(* Logix 5000 project; controller Final vendor 1 type 14 code 242 rev 32.11; software revision 32.00 *)

TASK MainTask (continuous, watchdog 500 ms) : MainProgram
TASK SafetyTask (periodic, rate 20 ms, priority 10, watchdog 20 ms, safety) : SafetyProgram

MODULES
   Local : vendor 1 type 14 code 242 (5069 0, rev 32.11)
      IO_002 : 5069-IF8 (5069 2, rev 2.1, StandardDataDriven RPI 100 ms)
      IO_001 : 5069-IF8 (5069 1, rev 2.1, StandardDataDriven RPI 100 ms)
      IO_003 : 5069-IF8 (5069 3, rev 2.1, StandardDataDriven RPI 100 ms)
      IO_006 : vendor 1 type 7 code 394 (5069 6, rev 2.1, StandardDataDriven RPI 5 ms)
      IO_004 : vendor 1 type 7 code 395 (5069 4, rev 2.1, StandardDataDriven RPI 5 ms)
      IO_005 : vendor 1 type 7 code 395 (5069 5, rev 2.1, StandardDataDriven RPI 5 ms)
      IO_007 : vendor 1 type 109 code 90 (5069 7, rev 3.1, StandardDataDriven RPI 80 ms)
      EN_001 : 1734-AENTR (Ethernet 192.168.1.60, rev 5.1, Output RPI 20 ms)
         EN_004 : 1734-485ASC (PointIO 3, rev 4.1, Output RPI 80 ms)
         EN_003 : vendor 1 type 35 code 16 (PointIO 2, rev 2.1, Input RPI 10 ms, Output RPI 20 ms)
         EN_002 : vendor 1 type 35 code 15 (PointIO 1, rev 2.1, Input RPI 10 ms)
END_MODULES

TYPE ASC_module_string :
STRUCT
   LEN : DINT;
   DATA : SINT[100];
END_STRUCT
END_TYPE

TYPE SensorType :   // To monitor the sensor readings, we use this data type
STRUCT
   CurrentValue : DINT;
   PreviousValue0 : DINT;
   PreviousValue1 : DINT;
   PreviousValue2 : DINT;
   PreviousValue3 : DINT;
   PreviousValue4 : DINT;
   PreviousValue5 : DINT;
   PreviousValue6 : DINT;
   PreviousValue7 : DINT;
   PreviousValue8 : DINT;
   PreviousValue9 : DINT;
   Mean10 : DINT;
   StanDev : DINT;
   State : DINT;
   Count : DINT;
   MeanStart : BOOL;
END_STRUCT
END_TYPE

TYPE String122 :
STRUCT
   LEN : DINT;
   DATA : SINT[122];
END_STRUCT
END_TYPE

VAR_GLOBAL   (* controller tags *)
   ACC_TIMER : DINT;
   ASC_module_Data : ASC_module_string;
   AT : BOOL;
   B0_Max : DINT;
   B0_Min : DINT;
   B1_Max : DINT;
   B1_Min : DINT;
   B3_Max : DINT;
   B3_Min : DINT;
   B_Check : BOOL;
   B_Checked : BOOL;
   B_NomCount : DINT := 24;
   B_Pres0 : SensorType := (CurrentValue := 15, PreviousValue0 := 15, PreviousValue1 := 15, PreviousValue2 := 15, PreviousValue3 := 15, PreviousValue4 := 15, PreviousValue5 := 15, PreviousValue6 := 15, PreviousValue7 := 15, PreviousValue8 := 15, PreviousValue9 := 15, Mean10 := 15, Count := 7, MeanStart := 1);   // Holds all values related to Brakes Pressure Sensor #0
   B_Pres1 : SensorType := (CurrentValue := 15, PreviousValue0 := 15, PreviousValue1 := 15, PreviousValue2 := 15, PreviousValue3 := 15, PreviousValue4 := 15, PreviousValue5 := 15, PreviousValue6 := 15, PreviousValue7 := 15, PreviousValue8 := 15, PreviousValue9 := 15, Mean10 := 15, Count := 7, MeanStart := 1);   // Holds all values related to Brakes Pressure Sensor #1
   B_Pres2 : SensorType := (CurrentValue := 15, PreviousValue0 := 15, PreviousValue1 := 15, PreviousValue2 := 15, PreviousValue3 := 15, PreviousValue4 := 15, PreviousValue5 := 15, PreviousValue6 := 15, PreviousValue7 := 15, PreviousValue8 := 15, PreviousValue9 := 15, Mean10 := 15, Count := 7, MeanStart := 1);   // Holds all values related to Brakes Pressure Sensor #2
   B_Pres3 : SensorType := (CurrentValue := 15, PreviousValue0 := 15, PreviousValue1 := 15, PreviousValue2 := 15, PreviousValue3 := 15, PreviousValue4 := 15, PreviousValue5 := 15, PreviousValue6 := 15, PreviousValue7 := 15, PreviousValue8 := 15, PreviousValue9 := 15, Mean10 := 15, Count := 7, MeanStart := 1);   // Holds all values related to Brakes Pressure Sensor #3
   B_Pres4 : SensorType := (CurrentValue := 15, PreviousValue0 := 15, PreviousValue1 := 15, PreviousValue2 := 15, PreviousValue3 := 15, PreviousValue4 := 15, PreviousValue5 := 15, PreviousValue6 := 15, PreviousValue7 := 15, PreviousValue8 := 15, PreviousValue9 := 15, Mean10 := 15, Count := 7, MeanStart := 1);   // Holds all values related to Brakes Pressure Sensor #4
   B_Pres5 : SensorType := (CurrentValue := 15, PreviousValue0 := 15, PreviousValue1 := 15, PreviousValue2 := 15, PreviousValue3 := 15, PreviousValue4 := 15, PreviousValue5 := 15, PreviousValue6 := 15, PreviousValue7 := 15, PreviousValue8 := 15, PreviousValue9 := 15, Mean10 := 15, Count := 7, MeanStart := 1);   // Holds all values related to Brakes Pressure Sensor #5
   B_Pres6 : SensorType := (CurrentValue := 15, PreviousValue0 := 15, PreviousValue1 := 15, PreviousValue2 := 15, PreviousValue3 := 15, PreviousValue4 := 15, PreviousValue5 := 15, PreviousValue6 := 15, PreviousValue7 := 15, PreviousValue8 := 15, PreviousValue9 := 15, Mean10 := 15, Count := 7, MeanStart := 1);   // Holds all values related to Brakes Pressure Sensor #6
   B_Pres7 : SensorType := (CurrentValue := 15, PreviousValue0 := 15, PreviousValue1 := 15, PreviousValue2 := 15, PreviousValue3 := 15, PreviousValue4 := 15, PreviousValue5 := 15, PreviousValue6 := 15, PreviousValue7 := 15, PreviousValue8 := 15, PreviousValue9 := 15, Mean10 := 15, Count := 7, MeanStart := 1);   // Holds all values related to Brakes Pressure Sensor #7
   B_Pres8 : SensorType := (CurrentValue := 15, PreviousValue0 := 15, PreviousValue1 := 15, PreviousValue2 := 15, PreviousValue3 := 15, PreviousValue4 := 15, PreviousValue5 := 15, PreviousValue6 := 15, PreviousValue7 := 15, PreviousValue8 := 15, PreviousValue9 := 15, Mean10 := 15, Count := 7, MeanStart := 1);   // Holds all values related to Brakes Pressure Sensor #8
   B_Pres9 : SensorType := (CurrentValue := 15, PreviousValue0 := 15, PreviousValue1 := 15, PreviousValue2 := 15, PreviousValue3 := 15, PreviousValue4 := 15, PreviousValue5 := 15, PreviousValue6 := 15, PreviousValue7 := 15, PreviousValue8 := 15, PreviousValue9 := 15, Mean10 := 15, Count := 7, MeanStart := 1);   // Holds all values related to Brakes Pressure Sensor #9
   B_Tem0 : SensorType := (CurrentValue := 92, PreviousValue0 := 92, PreviousValue1 := 92, PreviousValue2 := 92, PreviousValue3 := 92, PreviousValue4 := 92, PreviousValue5 := 92, PreviousValue6 := 92, PreviousValue7 := 92, PreviousValue8 := 92, PreviousValue9 := 92, Mean10 := 92, Count := 7, MeanStart := 1);   // Holds all values related to Brakes Temperature Sensor #0
   B_Tem1 : SensorType := (CurrentValue := 92, PreviousValue0 := 92, PreviousValue1 := 92, PreviousValue2 := 92, PreviousValue3 := 92, PreviousValue4 := 92, PreviousValue5 := 92, PreviousValue6 := 92, PreviousValue7 := 92, PreviousValue8 := 92, PreviousValue9 := 92, Mean10 := 92, Count := 7, MeanStart := 1);   // Holds all values related to Brakes Temperature Sensor #1
   Bat_Amp_State : DINT;
   BAT_FLAG : BOOL;
   Bat_Temp_State : DINT;
   Bat_Volt_State : DINT;
   BatCurrent_Pre : STRING;
   BatTemp_Pre : STRING;
   BATTERY_CHARGE : REAL := 104.21566;
   BATTERY_CURRENT : DINT;
   BATTERY_TEMP : REAL := 304.73172;
   BATTERY_VOLTAGE : REAL := 29.25294;
   BatteryA : REAL := 0.00112924;
   BatteryB : REAL := 0.000234108;
   BatteryC : REAL := 8.7755e-08;
   BatteryCommand : STRING := ':0102A0000EF6~';
   BatVoltage_Pre : STRING;
   BCount : DINT;
   bfr_SysSec : DINT := 58;
   BPCount : DINT;
   BRAKE_FLAG : BOOL;
   BRAKE_SUBSTATE1 : DINT;
   BRAKE_SUBSTATE2 : DINT;
   BRAKE_TIMER : FBD_TIMER;
   BRPM : DINT;
   BT : BOOL;
   C_Las0 : SensorType := (CurrentValue := 213, PreviousValue0 := 213, PreviousValue1 := 213, PreviousValue2 := 213, PreviousValue3 := 213, PreviousValue4 := 213, PreviousValue5 := 213, PreviousValue6 := 213, PreviousValue7 := 213, PreviousValue8 := 213, PreviousValue9 := 213, Mean10 := 213, Count := 7, MeanStart := 1);   // Holds all values related to Controls Laser Sensor #0
   C_Las1 : SensorType := (CurrentValue := 177, PreviousValue0 := 177, PreviousValue1 := 177, PreviousValue2 := 177, PreviousValue3 := 177, PreviousValue4 := 177, PreviousValue5 := 177, PreviousValue6 := 177, PreviousValue7 := 177, PreviousValue8 := 177, PreviousValue9 := 177, Mean10 := 177, Count := 7, MeanStart := 1);   // Holds all values related to Controls Laser Sensor #1
   CA : BOOL := 1;
   CB : BOOL;
   CC : BOOL;
   CD1 : BOOL := 1;
   CD2 : BOOL := 1;
   CD3 : BOOL := 1;
   COAST_TIMER : DINT;
   COAST_TONR : DINT;
   COMMAND : DINT := 1;
   COMN_FLAG : BOOL;
   ConversionResistance : REAL := 7533.3335;
   ConversionVoltage : REAL := 3.0;
   count : DINT;
   COUNT_LAS0 : DINT := 213;
   COUNT_LAS1 : DINT := 177;
   CP1 : BOOL := 1;
   CP2 : BOOL;
   CPX : BOOL;
   CT : BOOL;
   Current_OoR : BOOL := 1;
   CurrentState : DINT;
   CV : BOOL;
   DualStop : BOOL;
   EStop : BOOL;
   Initialized : DINT := 5380;
   InverseTemp : REAL := 0.003281575;
   LastValue : DINT;
   LastValue0 : DINT;
   LastValue1 : DINT;
   LenOut : SINT := 14;
   Limit1 : BOOL;
   Limit2 : BOOL;
   Local_TONR : FBD_TIMER;
   LogR : REAL := 8.927093;
   LSD_AA : BOOL;
   LSD_DR : BOOL;
   LSD_FR : BOOL;
   LSD_LC : DINT;
   LSD_PWR : BOOL;
   Mask : DINT := 16#0000_000f;
   my_TONR : FBD_TIMER;
   P_Check : DINT;
   P_Max : DINT;
   P_Mean : DINT;
   P_Min : DINT;
   P_NomCount : DINT := 20;
   P_Pres0 : SensorType := (CurrentValue := -16, PreviousValue0 := -16, PreviousValue1 := -16, PreviousValue2 := -16, PreviousValue3 := -16, PreviousValue4 := -16, PreviousValue5 := -16, PreviousValue6 := -16, PreviousValue7 := -16, PreviousValue8 := -16, PreviousValue9 := -16, Mean10 := -16, Count := 7, MeanStart := 1);   // Holds all values related to Pressure Pressure Sensor #0
   P_Pres0_FAILURE : BOOL;
   P_Pres1 : SensorType := (CurrentValue := -312, PreviousValue0 := -312, PreviousValue1 := -312, PreviousValue2 := -312, PreviousValue3 := -312, PreviousValue4 := -312, PreviousValue5 := -312, PreviousValue6 := -312, PreviousValue7 := -312, PreviousValue8 := -312, PreviousValue9 := -312, Count := 7);   // Holds all values related to Pressure Pressure Sensor #1
   P_Pres1_FAILURE : BOOL;
   P_Pres2 : SensorType := (CurrentValue := -312, PreviousValue0 := -312, PreviousValue1 := -312, PreviousValue2 := -312, PreviousValue3 := -312, PreviousValue4 := -312, PreviousValue5 := -312, PreviousValue6 := -312, PreviousValue7 := -312, PreviousValue8 := -312, PreviousValue9 := -312, Mean10 := -312, Count := 7, MeanStart := 1);   // Holds all values related to Pressure Pressure Sensor #2
   P_Pres2_FAILURE : BOOL;
   P_Pres3 : SensorType := (CurrentValue := -312, PreviousValue0 := -312, PreviousValue1 := -312, PreviousValue2 := -312, PreviousValue3 := -312, PreviousValue4 := -312, PreviousValue5 := -312, PreviousValue6 := -312, PreviousValue7 := -312, PreviousValue8 := -312, PreviousValue9 := -312, Mean10 := -312, Count := 7, MeanStart := 1);
   P_Pres3_FAILURE : BOOL;
   P_Pres4 : SensorType := (CurrentValue := -312, PreviousValue0 := -312, PreviousValue1 := -312, PreviousValue2 := -312, PreviousValue3 := -312, PreviousValue4 := -312, PreviousValue5 := -312, PreviousValue6 := -312, PreviousValue7 := -312, PreviousValue8 := -312, PreviousValue9 := -312, Mean10 := -312, Count := 7, MeanStart := 1);
   P_Pres4_FAILURE : BOOL;
   P_Tem0 : SensorType;   // Holds all values related to Pressure Temperature Sensor #0
   P_Tem0_FAILURE : BOOL;
   P_Tem1 : SensorType := (CurrentValue := 93, PreviousValue0 := 93, PreviousValue1 := 93, PreviousValue2 := 93, PreviousValue3 := 93, PreviousValue4 := 93, PreviousValue5 := 93, PreviousValue6 := 93, PreviousValue7 := 93, PreviousValue8 := 93, PreviousValue9 := 93, Mean10 := 93, Count := 7, MeanStart := 1);   // Holds all values related to Pressure Temperature Sensor #1
   P_Tem1_FAILURE : BOOL;
   P_Tem2 : SensorType := (CurrentValue := 93, PreviousValue0 := 93, PreviousValue1 := 93, PreviousValue2 := 93, PreviousValue3 := 93, PreviousValue4 := 93, PreviousValue5 := 93, PreviousValue6 := 93, PreviousValue7 := 93, PreviousValue8 := 93, PreviousValue9 := 93, Mean10 := 93, Count := 7, MeanStart := 1);
   P_Tem2_FAILURE : BOOL;
   P_Tem3 : SensorType := (CurrentValue := 93, PreviousValue0 := 93, PreviousValue1 := 93, PreviousValue2 := 93, PreviousValue3 := 93, PreviousValue4 := 93, PreviousValue5 := 93, PreviousValue6 := 93, PreviousValue7 := 93, PreviousValue8 := 93, PreviousValue9 := 93, Mean10 := 93, Count := 7, MeanStart := 1);
   P_Tem3_FAILURE : BOOL;
   P_Tem4 : SensorType := (CurrentValue := 93, PreviousValue0 := 93, PreviousValue1 := 93, PreviousValue2 := 93, PreviousValue3 := 93, PreviousValue4 := 93, PreviousValue5 := 93, PreviousValue6 := 93, PreviousValue7 := 93, PreviousValue8 := 93, PreviousValue9 := 93, Mean10 := 93, Count := 7, MeanStart := 1);
   P_Tem4_FAILURE : BOOL;
   POD_ACCELERATION : DINT;
   POD_DISTANCE : DINT := 1185672;
   POD_TIME : DINT[2] := ([0] := -1035744607, [1] := 205981);
   POD_VELOCITY : DINT;
   PREV_ACCELERATION : DINT;
   PREV_DISTANCE : DINT := 1185672;
   PREV_TIME : DINT[2] := ([0] := -1035744799);
   PREV_VELOCITY : DINT;
   PROP_FLAG : BOOL;
   PROP_STATE : BOOL;
   PROP_TNK_PRES : DINT;
   RcvRecord : SINT := 1;
   READY : BOOL;
   RxData : String122;
   RxID : SINT := 1;
   S_B_Pres0 : SensorType := (CurrentValue := 15, PreviousValue0 := 15, PreviousValue1 := 15, PreviousValue2 := 15, PreviousValue3 := 15, PreviousValue4 := 15, PreviousValue5 := 15, PreviousValue6 := 15, PreviousValue7 := 15, PreviousValue8 := 15, PreviousValue9 := 15, Mean10 := 15, Count := 7, MeanStart := 1);
   S_B_Pres1 : SensorType := (CurrentValue := 15, PreviousValue0 := 15, PreviousValue1 := 15, PreviousValue2 := 15, PreviousValue3 := 15, PreviousValue4 := 15, PreviousValue5 := 15, PreviousValue6 := 15, PreviousValue7 := 15, PreviousValue8 := 15, PreviousValue9 := 15, Mean10 := 15, Count := 7, MeanStart := 1);
   S_B_Pres2 : SensorType := (CurrentValue := 15, PreviousValue0 := 15, PreviousValue1 := 15, PreviousValue2 := 15, PreviousValue3 := 15, PreviousValue4 := 15, PreviousValue5 := 15, PreviousValue6 := 15, PreviousValue7 := 15, PreviousValue8 := 15, PreviousValue9 := 15, Mean10 := 15, Count := 7, MeanStart := 1);
   S_B_Pres3 : SensorType := (CurrentValue := 15, PreviousValue0 := 15, PreviousValue1 := 15, PreviousValue2 := 15, PreviousValue3 := 15, PreviousValue4 := 15, PreviousValue5 := 15, PreviousValue6 := 15, PreviousValue7 := 15, PreviousValue8 := 15, PreviousValue9 := 15, Mean10 := 15, Count := 7, MeanStart := 1);
   S_B_Pres4 : SensorType := (CurrentValue := 15, PreviousValue0 := 15, PreviousValue1 := 15, PreviousValue2 := 15, PreviousValue3 := 15, PreviousValue4 := 15, PreviousValue5 := 15, PreviousValue6 := 15, PreviousValue7 := 15, PreviousValue8 := 15, PreviousValue9 := 15, Mean10 := 15, Count := 7, MeanStart := 1);
   S_B_Pres5 : SensorType := (CurrentValue := 15, PreviousValue0 := 15, PreviousValue1 := 15, PreviousValue2 := 15, PreviousValue3 := 15, PreviousValue4 := 15, PreviousValue5 := 15, PreviousValue6 := 15, PreviousValue7 := 15, PreviousValue8 := 15, PreviousValue9 := 15, Mean10 := 15, Count := 7, MeanStart := 1);
   S_B_Pres6 : SensorType := (CurrentValue := 15, PreviousValue0 := 15, PreviousValue1 := 15, PreviousValue2 := 15, PreviousValue3 := 15, PreviousValue4 := 15, PreviousValue5 := 15, PreviousValue6 := 15, PreviousValue7 := 15, PreviousValue8 := 15, PreviousValue9 := 15, Mean10 := 15, Count := 7, MeanStart := 1);
   S_B_Pres7 : SensorType := (CurrentValue := 15, PreviousValue0 := 15, PreviousValue1 := 15, PreviousValue2 := 15, PreviousValue3 := 15, PreviousValue4 := 15, PreviousValue5 := 15, PreviousValue6 := 15, PreviousValue7 := 15, PreviousValue8 := 15, PreviousValue9 := 15, Mean10 := 15, Count := 7, MeanStart := 1);
   S_B_Pres8 : SensorType := (CurrentValue := 15, PreviousValue0 := 15, PreviousValue1 := 15, PreviousValue2 := 15, PreviousValue3 := 15, PreviousValue4 := 15, PreviousValue5 := 15, PreviousValue6 := 15, PreviousValue7 := 15, PreviousValue8 := 15, PreviousValue9 := 15, Mean10 := 15, Count := 7, MeanStart := 1);
   S_B_Pres9 : SensorType := (CurrentValue := 15, PreviousValue0 := 15, PreviousValue1 := 15, PreviousValue2 := 15, PreviousValue3 := 15, PreviousValue4 := 15, PreviousValue5 := 15, PreviousValue6 := 15, PreviousValue7 := 15, PreviousValue8 := 15, PreviousValue9 := 15, Mean10 := 15, Count := 7, MeanStart := 1);
   S_B_Tem0 : SensorType := (CurrentValue := 92, PreviousValue0 := 92, PreviousValue1 := 92, PreviousValue2 := 92, PreviousValue3 := 92, PreviousValue4 := 92, PreviousValue5 := 92, PreviousValue6 := 92, PreviousValue7 := 92, PreviousValue8 := 92, PreviousValue9 := 92, Mean10 := 92, Count := 7, MeanStart := 1);
   S_B_Tem1 : SensorType := (CurrentValue := 92, PreviousValue0 := 92, PreviousValue1 := 92, PreviousValue2 := 92, PreviousValue3 := 92, PreviousValue4 := 92, PreviousValue5 := 92, PreviousValue6 := 92, PreviousValue7 := 92, PreviousValue8 := 92, PreviousValue9 := 92, Mean10 := 92, Count := 7, MeanStart := 1);
   S_BAT_FLAG : BOOL;
   S_BatteryC : DINT;
   S_BatteryT : REAL := 304.73172;
   S_BatteryV : REAL := 29.25294;
   S_BRAKE_FLAG : BOOL;
   S_Brake_Sub1 : DINT;
   S_Brake_Sub2 : DINT;
   S_COMMAND : DINT := 1;
   S_COMN_FLAG : BOOL;
   S_COMN_STATE : BOOL := 1;
   S_P_Pres0 : SensorType := (CurrentValue := -16, PreviousValue0 := -16, PreviousValue1 := -16, PreviousValue2 := -16, PreviousValue3 := -16, PreviousValue4 := -16, PreviousValue5 := -16, PreviousValue6 := -16, PreviousValue7 := -16, PreviousValue8 := -16, PreviousValue9 := -16, Mean10 := -16, Count := 7, MeanStart := 1);
   S_P_Pres1 : SensorType := (CurrentValue := -312, PreviousValue0 := -312, PreviousValue1 := -312, PreviousValue2 := -312, PreviousValue3 := -312, PreviousValue4 := -312, PreviousValue5 := -312, PreviousValue6 := -312, PreviousValue7 := -312, PreviousValue8 := -312, PreviousValue9 := -312, Count := 7);
   S_P_Pres2 : SensorType := (CurrentValue := -312, PreviousValue0 := -312, PreviousValue1 := -312, PreviousValue2 := -312, PreviousValue3 := -312, PreviousValue4 := -312, PreviousValue5 := -312, PreviousValue6 := -312, PreviousValue7 := -312, PreviousValue8 := -312, PreviousValue9 := -312, Mean10 := -312, Count := 7, MeanStart := 1);
   S_P_Pres3 : SensorType := (CurrentValue := -312, PreviousValue0 := -312, PreviousValue1 := -312, PreviousValue2 := -312, PreviousValue3 := -312, PreviousValue4 := -312, PreviousValue5 := -312, PreviousValue6 := -312, PreviousValue7 := -312, PreviousValue8 := -312, PreviousValue9 := -312, Mean10 := -312, Count := 7, MeanStart := 1);
   S_P_Pres4 : SensorType := (CurrentValue := -312, PreviousValue0 := -312, PreviousValue1 := -312, PreviousValue2 := -312, PreviousValue3 := -312, PreviousValue4 := -312, PreviousValue5 := -312, PreviousValue6 := -312, PreviousValue7 := -312, PreviousValue8 := -312, PreviousValue9 := -312, Mean10 := -312, Count := 7, MeanStart := 1);
   S_P_Tem0 : SensorType;
   S_P_Tem1 : SensorType := (CurrentValue := 93, PreviousValue0 := 93, PreviousValue1 := 93, PreviousValue2 := 93, PreviousValue3 := 93, PreviousValue4 := 93, PreviousValue5 := 93, PreviousValue6 := 93, PreviousValue7 := 93, PreviousValue8 := 93, PreviousValue9 := 93, Mean10 := 93, Count := 7, MeanStart := 1);
   S_P_Tem2 : SensorType := (CurrentValue := 93, PreviousValue0 := 93, PreviousValue1 := 93, PreviousValue2 := 93, PreviousValue3 := 93, PreviousValue4 := 93, PreviousValue5 := 93, PreviousValue6 := 93, PreviousValue7 := 93, PreviousValue8 := 93, PreviousValue9 := 93, Mean10 := 93, Count := 7, MeanStart := 1);
   S_P_Tem3 : SensorType := (CurrentValue := 93, PreviousValue0 := 93, PreviousValue1 := 93, PreviousValue2 := 93, PreviousValue3 := 93, PreviousValue4 := 93, PreviousValue5 := 93, PreviousValue6 := 93, PreviousValue7 := 93, PreviousValue8 := 93, PreviousValue9 := 93, Mean10 := 93, Count := 7, MeanStart := 1);
   S_P_Tem4 : SensorType := (CurrentValue := 93, PreviousValue0 := 93, PreviousValue1 := 93, PreviousValue2 := 93, PreviousValue3 := 93, PreviousValue4 := 93, PreviousValue5 := 93, PreviousValue6 := 93, PreviousValue7 := 93, PreviousValue8 := 93, PreviousValue9 := 93, Mean10 := 93, Count := 7, MeanStart := 1);
   S_PROP_FLAG : BOOL;
   S_PROP_STATE : BOOL;
   S_STATE : DINT := 1;
   S_Switch : AB:5000_DO4:O:0;
   S_SysFail : BOOL := 1;
   SafetyTest : DINT := 6;
   StandardTest : DINT := 6;
   STATE : DINT := 1;
   STRIPE_COUNT : DINT := 389;
   STRIPE_ERROR0 : DINT := 176;
   STRIPE_ERROR1 : DINT := 212;
   Stripe_Reset : BOOL;
   sts_secStandard : DINT := 58;
   sts_SysSec : DINT := 58;
   SYSTEM_FAIL : BOOL;
   T_Mean : DINT;
   Temperature_OoR : BOOL;
   Test_TONR : FBD_TIMER;
   tmr_HB : TIMER := (PRE := 5000, ACC := 1420, EN := 1, TT := 1);   // TIMER Heartbeat
   tmr_XMIT : TIMER := (PRE := 5000, ACC := 3441, EN := 1, TT := 1);
   TOTAL_FAILURE : BOOL := 1;
   TRIGGER : BOOL[32] := ([0] := 1, [1] := 1);
   Tx_String : STRING[1] := ([0] := ':0102A0000EF6~');
   TxOut0 : SINT := 8;
   Voltage_OoR : BOOL := 1;
   WatchDog : FBD_TIMER;
   WD : BOOL;
   WD_State : DINT;
END_VAR

PROGRAM MainProgram   (* main routine MainRoutine *)
VAR
   ACC_TIMER : FBD_TIMER;
   COAST_TIMER : FBD_TIMER;
   SIMULATOR : FBD_TIMER;
END_VAR

ROUTINE A01_Initialize   (* structured text *)
// Initializes the values of all tags
   JSR(Initial_B_Pres0); //Initialize Brake Pressure Sensor 0
   JSR(Initial_B_Pres1); //Initialize Brake Pressure Sensor 1
   JSR(Initial_B_Pres2); //Initialize Brake Pressure Sensor 2
   JSR(Initial_B_Pres3); //Initialize Brake Pressure Sensor 3
   JSR(Initial_B_Pres4); //Initialize Brake Pressure Sensor 4
   JSR(Initial_B_Pres5); //Initialize Brake Pressure Sensor 5
   JSR(Initial_B_Pres6); //Initialize Brake Pressure Sensor 6
   JSR(Initial_B_Pres7); //Initialize Brake Pressure Sensor 7
   JSR(Initial_B_Pres8); //Initialize Brake Pressure Sensor 8
   JSR(Initial_B_Pres9); //Initialize Brake Pressure Sensor 9
   JSR(Initial_B_Tem0); //Initialize Brake Temperature Sensor 0
   JSR(Initial_B_Tem1); //Initialize Brake Temperature Sensor 1
   Local:4:O.Pt02.Data := 1; //Set NOV-1 & NOV-2 to ON
   Local:4:O.Pt03.Data := 0; //Set NCV-1 & NCV-2 to ON
   B_NomCount := 24; //Assume all brakes sensors are working
   //Brakes Initialization Sequence complete
   
   JSR(Initial_C_Las0); //Initialize Controls Laser Sensor 0
   JSR(Initial_C_Las1);  //Initialize Controls Laser Sensor 1
    //Controls Initialization Sequence complete
   
   JSR(Initial_P_Pres0); //Initialize Propulsion Pressure Sensor 0
   JSR(Initial_P_Pres1); //Initialize Propulsion Pressure Sensor 1
   JSR(Initial_P_Pres2); //Initialize Propulsion Pressure Sensor 2
   JSR(Initial_P_Pres3); //Initialize Propulsion Pressure Sensor 3
   JSR(Initial_P_Pres4); //Initialize Propulsion Pressure Sensor 4
   JSR(Initial_P_Tem1); //Initialize Propulsion Temperature Sensor 1
   JSR(Initial_P_Tem2); //Initialize Propulsion Temperature Sensor 2
   JSR(Initial_P_Tem3); //Initialize Propulsion Temperature Sensor 3
   JSR(Initial_P_Tem4); //Initialize Propulsion Temperature Sensor 4
   Local:5:O.Pt00.Data := 1; //Set S-1 (NOV) to ON
   Local:4:O.Pt00.Data := 0; //Set S-2 (NCV) to OFF
   Local:4:O.Pt01.Data := 0; //Set S-3 (NCV) to OFF
   P_NomCount := 18; //Assume all propulsion sensors are working
   //Propulsion Initialization Sequence complete
   
   BATTERY_CURRENT := 0; //Initialize Battery Current
   BATTERY_TEMP := 0; //Initialize Battery Temperature
   BATTERY_VOLTAGE := 0; //Initialize Battery Voltage
   //Power Initialization complete
   
   Local:5:O.Pt01.Data := 1; //Actuator Up
   Local:5:O.Pt02.Data := 1; //Motor Direction
   Local:5:O.Pt03.Data := 0; //Motor Power
   //Low-speed Drive Initialization Complete
   
   STRIPE_ERROR0 := 0; //Measure error in laser 0
   STRIPE_ERROR1 := 0; //Measure error in laser 1
   STRIPE_COUNT := 0; //Measure retroreflective stripes passed
   POD_TIME[0] := 0; //Pod time initalized to 0
   POD_DISTANCE := 0; //Measure distance of pod from start of the tube
   POD_VELOCITY := 0; //Measure velocity of pod
   POD_ACCELERATION := 0; //Measure acceleration of pod
   READY := 0; //Tells when pod is ready to launch
   PROP_TNK_PRES := 0; //Average pressure of all propulsion tanks
   PROP_STATE := 0; //State of propulsion system: 0 = Nominal; 1 = Failure
   BRAKE_SUBSTATE1 := 0; //State of brake subsystem 1: 0 = Nominal; 1 = Failure
   BRAKE_SUBSTATE2 := 0; //State of brake subsystem 2: 0 = Nominal; 1 = Failure
   PROP_FLAG := 0; //Identifier for integrity of propulsion system: 0 = Nominal; 1 = Failure
   BRAKE_FLAG := 0; //Identifier for integrity of brake system: 0 = Nominal; 1 = Failure
   COMN_FLAG := 0; //Identifier for integrity of communication system: 0 = Nominal; 1 = Failure
   BAT_FLAG := 0; //Identifier for integrity of battery system: 0 = Nominal; 1 = Failure
   SYSTEM_FAIL := 0; //Identifier for integrity of entire system: 0 = Nominal; 1 = Failure
   STATE := 1; //Set state to Idle
   COMMAND := 1; //Set command to IDLE
   CD1 := 0;
   CD2 := 0;
   CD3 := 0;
   CA := 0;
   AT := 0;
   BT := 0;
   CT := 0;
   CP1 := 0;
   CP2 := 0;
   CV := 0;
   //State checks initialized
   WD_State := 0;
   WatchDog.PRE := 2700000;
   WatchDog.TimerEnable := 1;
   WatchDog.Reset := 0;
   TONR(WatchDog); //Timer that switches to Emergency Shutdown if no state changes are observed for 45 minutes
   B_Check := 0;
   B_Checked := 0;
   P_Check := 0;
   Initialized := 5380; //Initialization complete
END_ROUTINE

ROUTINE A02_Update   (* structured text *)
// Updates all sensor value tags
   /*IO Link : Associated parameter
   Local:1:I.Ch00.Data : B_Pres0.CurrentValue
   Local:1:I.Ch01.Data : B_Pres1.CurrentValue
   Local:1:I.Ch02.Data : B_Pres2.CurrentValue
   Local:1:I.Ch03.Data : B_Pres3.CurrentValue
   Local:1:I.Ch04.Data : B_Pres4.CurrentValue
   Local:1:I.Ch05.Data : B_Pres5.CurrentValue
   Local:1:I.Ch06.Data : B_Pres6.CurrentValue
   Local:1:I.Ch07.Data : B_Pres7.CurrentValue
   Local:2:I.Ch00.Data : B_Pres8.CurrentValue
   Local:2:I.Ch01.Data : B_Pres9.CurrentValue
   Local:2:I.Ch02.Data : B_Tem0.CurrentValue*
   Local:2:I.Ch03.Data : B_Tem1.CurrentValue*
   Local:2:I.Ch04.Data : P_Pres0.CurrentValue
   Local:2:I.Ch05.Data : Battery Voltage
   Local:2:I.Ch06.Data : Battery Temperature
   Local:2:I.Ch07.Data : //Battery Current*
   Local:3:I.Ch00.Data : P_Pres1.CurrentValue
   Local:3:I.Ch01.Data : P_Pres2.CurrentValue
   Local:3:I.Ch02.Data : P_Pres3.CurrentValue
   Local:3:I.Ch03.Data : P_Pres4.CurrentValue
   Local:3:I.Ch04.Data : P_Tem1.CurrentValue
   Local:3:I.Ch05.Data : P_Tem2.CurrentValue
   Local:3:I.Ch06.Data : P_Tem3.CurrentValue
   Local:3:I.Ch07.Data : P_Tem4.CurrentValue
   Local:4:O.Pt.00.Data : S-2 (propulsion)
   Local:4:O.Pt.01.Data : S-3 (propulsion)
   Local:4:O.Pt.02.Data : NOV-1 & NOV-2 (brakes)
   Local:4:O.Pt.03.Data : NCV-1 & NCV-2 (brakes)
   Local:5:O.Pt.00.Data : S-1 (propulsion)
   Local:5:O.Pt.01.Data : Actuator Direction (LSD)
   Local:5:O.Pt.02.Data : Motor Direction (LSD)
   Local:5:O.Pt.03.Data : Motor Power (LSD)
   Local:6:I.Pt00.Data : L-1 (propulsion)*
   Local:6:I.Pt01.Data : L-2 (propulsion)*
   Local:6:I.Pt02.Data : <unassigned>
   Local:6:I.Pt03.Data : <unassigned>
   Local:6:I.Pt04.Data : <unassigned>
   Local:6:I.Pt05.Data : <unassigned>
   Local:7:I.Counter00.Count : C_Las0.Count
   Local:7:I.Counter01.Count : C_Las1.Count
   EN_001:1:I.Pt00Data : <unassigned>
   EN_001:1:I.Pt01Data : <unassigned>
   EN_001:1:I.Pt02Data : <unassigned>
   EN_001:1:I.Pt03Data : <unassigned>
   EN_001:1:I.Pt04Data : <unassigned>
   EN_001:1:I.Pt05Data : <unassigned>
   EN_001:1:I.Pt06Data : <unassigned>
   EN_001:1:I.Pt07Data : <unassigned>
   EN_001:2:O.Pt00Data : <unassigned>
   EN_001:2:O.Pt01Data : <unassigned>
   EN_001:2:O.Pt02Data : <unassigned>
   EN_001:2:O.Pt03Data : <unassigned>
   EN_001:2:O.Pt04Data : <unassigned>
   EN_001:2:O.Pt05Data : <unassigned>
   EN_001:2:O.Pt06Data : <unassigned>
   EN_001:2:O.Pt07Data : <unassigned>
   EN_001:3:I.Data : <unassigned>
   EN_001:3:I.Length : <unassigned>
   EN_001:3:O.Data : <unassigned>
   //Safety Modules disconnected
   */
   
   JSR(Update_B_Pres0); //Updates associated variables of Brake Pressure sensor 0
   JSR(Update_B_Pres1); //Updates associated variables of Brake Pressure sensor 1
   JSR(Update_B_Pres2); //Updates associated variables of Brake Pressure sensor 2
   JSR(Update_B_Pres3); //Updates associated variables of Brake Pressure sensor 3
   JSR(Update_B_Pres4); //Updates associated variables of Brake Pressure sensor 4
   JSR(Update_B_Pres5); //Updates associated variables of Brake Pressure sensor 5
   JSR(Update_B_Pres6); //Updates associated variables of Brake Pressure sensor 6
   JSR(Update_B_Pres7); //Updates associated variables of Brake Pressure sensor 7
   JSR(Update_B_Pres8); //Updates associated variables of Brake Pressure sensor 8
   JSR(Update_B_Pres9); //Updates associated variables of Brake Pressure sensor 9
   JSR(Update_B_Tem0); //Updates associated variables of Brake Temperature sensor 0
   JSR(Update_B_Tem1); //Updates associated variables of Brake Temperature sensor 1
   //Brakes sensors up-to-date
   
   JSR(Update_P_Pres0); //Updates associated variables of Propulsion Pressure sensor 1
   JSR(Update_P_Pres1); //Updates associated variables of Propulsion Pressure sensor 1
   JSR(Update_P_Pres2); //Updates associated variables of Propulsion Pressure sensor 2
   JSR(Update_P_Pres3); //Updates associated variables of Propulsion Pressure sensor 3
   JSR(Update_P_Pres4); //Updates associated variables of Propulsion Pressure sensor 4
   JSR(Update_P_Tem1); //Updates associated variables of Propulsion Temperature sensor 1
   JSR(Update_P_Tem2); //Updates associated variables of Propulsion Temperature sensor 2
   JSR(Update_P_Tem3); //Updates associated variables of Propulsion Temperature sensor 3
   JSR(Update_P_Tem4); //Updates associated variables of Propulsion Temperature sensor 4
   JSR(Update_Limit1); //Updates limit switch 1 position
   JSR(Update_Limit2); //Updates limit switch 2 position
   //Propulsion sensors up-to-date
   
   JSR(Update_C_Las0); //Updates associated variables of Controls Laser sensor 0
   JSR(Update_C_Las1); //Updates associated variables of Controls Laser sensor 1
   //Controls sensors up-to-date
   
   JSR(Update_Battery_Temp); //Updates battery pack temperature
   JSR(Update_Battery_Volt); //Updates battery pack voltage
   JSR(Update_Battery_Amp);  //Updates battery pack current
   //Power parameters up-to-date
   
   JSR(MiniMax); //Sets minimum and maximum values of braking thresholds
   JSR(NomCheck_B1); //Nominality Check for Brakes
   JSR(NomCheck_P1); //Nominality Check for Propulsion
   JSR(NomCheck_BT); //Nominality Check for Battery
   //Local:4:O.Pt00.Data := Local:4:O.Pt01.Data; //Confirm both valves are same state
END_ROUTINE

ROUTINE A03_Process   (* structured text *)
// Processes input data
   //High Speed Counter interface
   GSV(WallClockTime,,CurrentValue,POD_TIME[0]); //units microseconds
   if Stripe_Reset then
   	LastValue0 := Local:7:I.Counter00.Count;
   	LastValue1 := Local:7:I.Counter01.Count;
   	STRIPE_ERROR0 := 0;
   	STRIPE_ERROR1 := 0;
   	STRIPE_COUNT := 0;
   	POD_DISTANCE := 3048 * STRIPE_COUNT;
   end_if;
   COUNT_LAS0 := C_Las0.CurrentValue - LastValue0;
   COUNT_LAS1 := C_Las1.CurrentValue - LastValue1;
   
   if (COUNT_LAS0 + STRIPE_ERROR0) > (COUNT_LAS1 + STRIPE_ERROR1) then
   STRIPE_ERROR1 := STRIPE_ERROR1 + 1;
   STRIPE_COUNT := COUNT_LAS0 + STRIPE_ERROR0;
   POD_DISTANCE := 3048 * STRIPE_COUNT; //units cm
   POD_VELOCITY := 3048 * Local:7:I.Counter00.Frequency; //(POD_DISTANCE - PREV_DISTANCE)/(100000*(POD_TIME[0] - PREV_TIME[0])); //units cm/s
   POD_ACCELERATION := 3048 * Local:7:I.Counter00.Accel; //(POD_VELOCITY - PREV_VELOCITY)/(POD_TIME[0] - PREV_TIME[0]); //units cm/s2
   
   elsif (COUNT_LAS0 + STRIPE_ERROR0) < (COUNT_LAS1 + STRIPE_ERROR1) then
   STRIPE_ERROR0 := STRIPE_ERROR0 + 1;
   STRIPE_COUNT := COUNT_LAS1 + STRIPE_ERROR1;
   POD_DISTANCE := 3048 * STRIPE_COUNT; //units cm
   POD_VELOCITY := 3048 * Local:7:I.Counter01.Frequency; //(POD_DISTANCE - PREV_DISTANCE)/(100000*(POD_TIME[0] - PREV_TIME[0])); //units cm/s
   POD_ACCELERATION := 3048 * Local:7:I.Counter01.Accel; //(POD_VELOCITY - PREV_VELOCITY)/(POD_TIME[0] - PREV_TIME[0]); //units cm/s2
   end_if;
   
   //Process Data part 2
END_ROUTINE

ROUTINE A04_State   (* structured text *)
// Updates the state of the pod
   JSR(Check_Distance_1); //Checks if POD_DISTANCE >= 3000 cm
   JSR(Check_Distance_2); //Checks if POD_DISTANCE >= 80000 cm
   JSR(Check_Distance_3); //Checks if POD_DISTANCE >= 125000 cm
   JSR(Check_TankPres_1); //Checks if PROP_TNK_PRES >= 200 PSI
   JSR(Check_TankPres_2); //Checks if PROP_TNK_PRES <= 100 PSI
   JSR(Check_PodAcc_1); //Checks if POD_ACCELERATION <= 0 cm/s2
   JSR(Check_PodVel_1); //Checks if POD_VELOCITY >= 2862 cm/s
   JSR(Check_AccTimer); // Checks if ACC_TIMER >= 7.7 sec
   JSR(Check_CoastTimer); //Checks if COAST_TIMER >= 10 sec
   JSR(Check_BrakeTimer); //Checks if BRAKE_TIMER >= 10 sec
   JSR(Check_WatchDog); //Checks if Watchdog is done
END_ROUTINE

ROUTINE A05_Actions   (* structured text *)
// Performs the state actions of the pod
   if WD then
   	JSR(B10_EmergencyShutdown);
   elsif WD_State <> STATE then
   	WD_State := STATE;
   	WatchDog.Reset := 1;
   	TONR(WatchDog);
   end_if;
   
   case STATE of
   	1: JSR(B01_Idle);
   	2: JSR(B02_SystemCheck);
   	3: JSR(B03_Armed);
   	4: JSR(B04_Acceleration);
   	5: JSR(B05_Coast);
   	6: JSR(B06_Brake);
   	7: JSR(B07_Stop);
   	8: JSR(B08_Crawl);
   	9: JSR(B09_End);
   	10: JSR(B10_EmergencyShutdown);
   	11: JSR(B11_Safe);
   end_case;
   
   //Command legend
   //1 - IDLE
   //2 - BEGIN
   //3 - ARM
   //4 - LAUNCH
   //5 - <unassigned>
   //6 - <unassigned>
   //7 - STOP
   //8 - CRAWL
   //9 - END
   //10 - EGSD
END_ROUTINE

ROUTINE B01_Idle   (* structured text *)
   //Check for command receieved
   if COMMAND = 2 then
   	STATE := 2; //System Check
   end_if;
   
   if COMMAND = 9 then
   	STATE := 9; //End
   end_if;
   
   if COMMAND = 10 then
   	STATE := 1; //Idle
   end_if;
END_ROUTINE

ROUTINE B02_SystemCheck   (* structured text *)
   if B_NomCount <> 24 then
   	JSR(FaultTest_B);
   end_if;
   
   if P_NomCount <> 18 then
   	JSR(FaultTest_P);
   end_if;
   
   if COMMAND = 3 then
   	STATE := 3; //Armed
   end_if;
   
   if COMMAND = 1 then
   	STATE := 1; //Idle
   end_if;
   
   if COMMAND = 10 then
   	STATE := 1; //Emergency Shutdown
   end_if;
   
   if B_Check then
   Local:4:O.Pt02.Data := 0; //Engaging brakes
   Local:4:O.Pt03.Data := 0; //Brakes engaged
   else
   Local:4:O.Pt02.Data := 1; //Disengaging brakes
   	Test_TONR.PRE := 5000;
   	Test_TONR.TimerEnable := 1;
   	Test_TONR.Reset := 0;
   	TONR(Test_TONR);
   	if Test_TONR.DN then
   	Local:4:O.Pt03.Data := 1; //Brakes disengaged
   	Test_TONR.Reset := 1;
   	TONR(Test_TONR);
   	end_if;
   end_if;
END_ROUTINE

ROUTINE B03_Armed   (* structured text *)
   if COMMAND = 4 then
   	STATE := 4; //Acceleration
   end_if;
   
   if COMMAND = 8 then
   	STATE := 8; //Crawl
   end_if;
   
   if COMMAND = 10 then
   	STATE := 10; //Emergency Shutdown
   end_if;
END_ROUTINE

ROUTINE B04_Acceleration   (* structured text *)
   ACC_TIMER.PRE := 5000;
   ACC_TIMER.TimerEnable := 1;
   ACC_TIMER.Reset := 0;
   TONR(ACC_TIMER);
   
   Local:4:O.Pt00.Data := 1;
   Local:4:O.Pt01.Data := 1; //Activate Propulsion
   
   if CP1 OR CA OR AT OR CV then //PROP_TNK_PRES <= 200 PSI or Accleration < 0 or Velocity >= 60
   	STATE := 5; //Coast
   end_if;
   
   if COMMAND = 10 then
   	STATE := 10; //Emergency Shutdown
   end_if;
END_ROUTINE

ROUTINE B05_Coast   (* structured text *)
   COAST_TIMER.PRE := 20000; //
   COAST_TIMER.TimerEnable := 1;
   COAST_TIMER.Reset := 0;
   TONR(COAST_TIMER); //Coast timer initialized
   
   Local:4:O.Pt00.Data := 0;
   Local:4:O.Pt01.Data := 0; //Propulsion disengaged
   
   if CP2 then
   	Local:5:O.Pt00.Data := 0; //Relief pressure valve open
   end_if;
   
   if CD2 OR CT OR (COMMAND = 7) then
   	STATE := 6; //Brake
   end_if;
   
   if COMMAND = 10 then
   	STATE := 10; //Emergency Shutdown
   end_if;
END_ROUTINE

ROUTINE B06_Brake   (* structured text *)
   BRAKE_TIMER.PRE := 10000;
   BRAKE_TIMER.TimerEnable := 1;
   BRAKE_TIMER.Reset := 0;
   TONR(BRAKE_TIMER); //Brake timer initialized
   
   Local:5:O.Pt00.Data := 1; //Relief pressure valve closed
   Local:4:O.Pt02.Data := 0; //Engaging brakes
   Local:4:O.Pt03.Data := 0; //Brakes engaged
   
   if POD_VELOCITY = 0 or BT then
   	STATE := 7; //Stop
   end_if;
   
   if (COMMAND = 10) OR (NOT CA) then //If POD_ACCLERATION > 0
   	STATE := 10; //Emergency Shutdown
   end_if;
END_ROUTINE

ROUTINE B07_Stop   (* structured text *)
   Local:4:O.Pt02.Data := 1; //Disengaging brakes
   	Local_TONR.PRE := 2000;
   	Local_TONR.TimerEnable := 1;
   	Local_TONR.Reset := 0;
   	TONR(Local_TONR);
   if Local_TONR.DN then
   	Local:4:O.Pt03.Data := 1; //Brakes disengaged
   end_if;
   
   if COMMAND = 8 then
   STATE := 8; //Crawl
   end_if;
   
   if COMMAND = 9 then
   STATE := 9; //End
   end_if;
   
   if COMMAND = 10 then
   	STATE := 10; //Emergency Shutdown
   end_if;
END_ROUTINE

ROUTINE B08_Crawl   (* structured text *)
   Local:5:O.Pt01.Data := 0; //Actuator down
   
   my_TONR.PRE := 3000;
   my_TONR.TimerEnable := 1;
   my_TONR.Reset := 0;
   TONR(my_TONR);
   if my_TONR.DN then
   	Local:5:O.Pt03.Data := 1; //Motor Power
   	my_TONR.Reset := 1;
   TONR(my_TONR);
   else
   	Local:5:O.Pt03.Data := 0; //Motor Power
   end_if;
   
   if CD3 OR (COMMAND = 7) then
   	Local:5:O.Pt01.Data := 1; //Actuator up
   	Local:5:O.Pt03.Data := 0; //Motor Power
   	STATE := 6; //Stop
   end_if;
END_ROUTINE

ROUTINE B09_End   (* structured text *)
   Local:4:O.Pt02.Data := 0; //Brake tanks pressure relieving
   Local:4:O.Pt03.Data := 1; //Brake tanks pressure relieved
   //Reached end of tube
END_ROUTINE

ROUTINE B10_EmergencyShutdown   (* structured text *)
   if CA then
   	Local:4:O.Pt00.Data := 0; //Closing propulsion tanks
   	Local:4:O.Pt01.Data := 0; //Propulsion tanks closed
   	Local:5:O.Pt01.Data := 1; //Actuator up
   	Local:5:O.Pt03.Data := 0; //Motor power off
   end_if;
   Local:4:O.Pt02.Data := 0;
   Local:4:O.Pt03.Data := 0; //Brakes activated
   
   if CP2 then
   	STATE := 7; //Stop
   else
   	Local:4:O.Pt00.Data := 0; //Relief pressure valve
   	STATE := 7; //Stop
   end_if;
END_ROUTINE

ROUTINE B11_Safe   (* structured text *)
   
END_ROUTINE

ROUTINE Check_AccTimer   (* structured text *)
   if ACC_TIMER.DN then
   	AT := 1;
   end_if;
END_ROUTINE

ROUTINE Check_BrakeTimer   (* structured text *)
   if BRAKE_TIMER.DN then
   	BT := 1;
   end_if;
END_ROUTINE

ROUTINE Check_CoastTimer   (* structured text *)
   if COAST_TIMER.DN then
   	CT := 1;
   	end_if;
END_ROUTINE

ROUTINE Check_Distance_1   (* structured text *)
   if POD_DISTANCE >= 3000 then
   	CD1 := 1;
   end_if;
END_ROUTINE

ROUTINE Check_Distance_2   (* structured text *)
   if POD_DISTANCE >= 80000 then
   	CD2 := 1;
   end_if;
END_ROUTINE

ROUTINE Check_Distance_3   (* structured text *)
   if POD_DISTANCE >= 125000 then
   	CD3 := 1;
   end_if;
END_ROUTINE

ROUTINE Check_PodAcc_1   (* structured text *)
   if POD_ACCELERATION <= 0 then
   	CA := 1;
   end_if;
END_ROUTINE

ROUTINE Check_PodVel_1   (* structured text *)
   if POD_VELOCITY >= 1117.6 then //25 mph
   	CV := 1;
   end_if;
END_ROUTINE

ROUTINE Check_TankPres_1   (* structured text *)
   if (P_Pres1.CurrentValue + P_Pres2.CurrentValue + P_Pres3.CurrentValue + P_Pres4.CurrentValue) <= 20 then
   	CP1 := 1;
   end_if;
END_ROUTINE

ROUTINE Check_TankPres_2   (* structured text *)
   if (P_Pres1.CurrentValue + P_Pres2.CurrentValue + P_Pres3.CurrentValue + P_Pres4.CurrentValue) <= 10 then
   	CP2 := 1;
   end_if;
END_ROUTINE

ROUTINE Check_WatchDog   (* structured text *)
   if WatchDog.DN then
   	WD := 1;
   end_if;
END_ROUTINE

ROUTINE FaultTest_B   (* structured text *)
   
END_ROUTINE

ROUTINE FaultTest_P   (* structured text *)
   
END_ROUTINE

ROUTINE Initial_B_Pres0   (* structured text *)
   B_Pres0.CurrentValue := 0;
   B_Pres0.PreviousValue0 := 0;
   B_Pres0.PreviousValue1 := 0;
   B_Pres0.PreviousValue2 := 0;
   B_Pres0.PreviousValue3 := 0;
   B_Pres0.PreviousValue4 := 0;
   B_Pres0.PreviousValue5 := 0;
   B_Pres0.PreviousValue6 := 0;
   B_Pres0.PreviousValue7 := 0;
   B_Pres0.PreviousValue8 := 0;
   B_Pres0.PreviousValue9 := 0;
   B_Pres0.Count := 0;
   B_Pres0.Mean10 := 0;
   B_Pres0.StanDev := 0;
   B_Pres0.State := 0;
   B_Pres0.MeanStart := 0;
END_ROUTINE

ROUTINE Initial_B_Pres1   (* structured text *)
   B_Pres1.CurrentValue := 0;
   B_Pres1.PreviousValue0 := 0;
   B_Pres1.PreviousValue1 := 0;
   B_Pres1.PreviousValue2 := 0;
   B_Pres1.PreviousValue3 := 0;
   B_Pres1.PreviousValue4 := 0;
   B_Pres1.PreviousValue5 := 0;
   B_Pres1.PreviousValue6 := 0;
   B_Pres1.PreviousValue7 := 0;
   B_Pres1.PreviousValue8 := 0;
   B_Pres1.PreviousValue9 := 0;
   B_Pres1.Count := 0;
   B_Pres1.Mean10 := 0;
   B_Pres1.StanDev := 0;
   B_Pres1.State := 0;
   B_Pres1.MeanStart := 0;
END_ROUTINE

ROUTINE Initial_B_Pres2   (* structured text *)
   B_Pres2.CurrentValue := 0;
   B_Pres2.PreviousValue0 := 0;
   B_Pres2.PreviousValue1 := 0;
   B_Pres2.PreviousValue2 := 0;
   B_Pres2.PreviousValue3 := 0;
   B_Pres2.PreviousValue4 := 0;
   B_Pres2.PreviousValue5 := 0;
   B_Pres2.PreviousValue6 := 0;
   B_Pres2.PreviousValue7 := 0;
   B_Pres2.PreviousValue8 := 0;
   B_Pres2.PreviousValue9 := 0;
   B_Pres2.Count := 0;
   B_Pres2.Mean10 := 0;
   B_Pres2.StanDev := 0;
   B_Pres2.State := 0;
   B_Pres2.MeanStart := 0;
END_ROUTINE

ROUTINE Initial_B_Pres3   (* structured text *)
   B_Pres3.CurrentValue := 0;
   B_Pres3.PreviousValue0 := 0;
   B_Pres3.PreviousValue1 := 0;
   B_Pres3.PreviousValue2 := 0;
   B_Pres3.PreviousValue3 := 0;
   B_Pres3.PreviousValue4 := 0;
   B_Pres3.PreviousValue5 := 0;
   B_Pres3.PreviousValue6 := 0;
   B_Pres3.PreviousValue7 := 0;
   B_Pres3.PreviousValue8 := 0;
   B_Pres3.PreviousValue9 := 0;
   B_Pres3.Count := 0;
   B_Pres3.Mean10 := 0;
   B_Pres3.StanDev := 0;
   B_Pres3.State := 0;
   B_Pres3.MeanStart := 0;
END_ROUTINE

ROUTINE Initial_B_Pres4   (* structured text *)
   B_Pres4.CurrentValue := 0;
   B_Pres4.PreviousValue0 := 0;
   B_Pres4.PreviousValue1 := 0;
   B_Pres4.PreviousValue2 := 0;
   B_Pres4.PreviousValue3 := 0;
   B_Pres4.PreviousValue4 := 0;
   B_Pres4.PreviousValue5 := 0;
   B_Pres4.PreviousValue6 := 0;
   B_Pres4.PreviousValue7 := 0;
   B_Pres4.PreviousValue8 := 0;
   B_Pres4.PreviousValue9 := 0;
   B_Pres4.Count := 0;
   B_Pres4.Mean10 := 0;
   B_Pres4.StanDev := 0;
   B_Pres4.State := 0;
   B_Pres4.MeanStart := 0;
END_ROUTINE

ROUTINE Initial_B_Pres5   (* structured text *)
   B_Pres5.CurrentValue := 0;
   B_Pres5.PreviousValue0 := 0;
   B_Pres5.PreviousValue1 := 0;
   B_Pres5.PreviousValue2 := 0;
   B_Pres5.PreviousValue3 := 0;
   B_Pres5.PreviousValue4 := 0;
   B_Pres5.PreviousValue5 := 0;
   B_Pres5.PreviousValue6 := 0;
   B_Pres5.PreviousValue7 := 0;
   B_Pres5.PreviousValue8 := 0;
   B_Pres5.PreviousValue9 := 0;
   B_Pres5.Count := 0;
   B_Pres5.Mean10 := 0;
   B_Pres5.StanDev := 0;
   B_Pres5.State := 0;
   B_Pres5.MeanStart := 0;
END_ROUTINE

ROUTINE Initial_B_Pres6   (* structured text *)
   B_Pres6.CurrentValue := 0;
   B_Pres6.PreviousValue0 := 0;
   B_Pres6.PreviousValue1 := 0;
   B_Pres6.PreviousValue2 := 0;
   B_Pres6.PreviousValue3 := 0;
   B_Pres6.PreviousValue4 := 0;
   B_Pres6.PreviousValue5 := 0;
   B_Pres6.PreviousValue6 := 0;
   B_Pres6.PreviousValue7 := 0;
   B_Pres6.PreviousValue8 := 0;
   B_Pres6.PreviousValue9 := 0;
   B_Pres6.Count := 0;
   B_Pres6.Mean10 := 0;
   B_Pres6.StanDev := 0;
   B_Pres6.State := 0;
   B_Pres6.MeanStart := 0;
END_ROUTINE

ROUTINE Initial_B_Pres7   (* structured text *)
   B_Pres7.CurrentValue := 0;
   B_Pres7.PreviousValue0 := 0;
   B_Pres7.PreviousValue1 := 0;
   B_Pres7.PreviousValue2 := 0;
   B_Pres7.PreviousValue3 := 0;
   B_Pres7.PreviousValue4 := 0;
   B_Pres7.PreviousValue5 := 0;
   B_Pres7.PreviousValue6 := 0;
   B_Pres7.PreviousValue7 := 0;
   B_Pres7.PreviousValue8 := 0;
   B_Pres7.PreviousValue9 := 0;
   B_Pres7.Count := 0;
   B_Pres7.Mean10 := 0;
   B_Pres7.StanDev := 0;
   B_Pres7.State := 0;
   B_Pres7.MeanStart := 0;
END_ROUTINE

ROUTINE Initial_B_Pres8   (* structured text *)
   B_Pres8.CurrentValue := 0;
   B_Pres8.PreviousValue0 := 0;
   B_Pres8.PreviousValue1 := 0;
   B_Pres8.PreviousValue2 := 0;
   B_Pres8.PreviousValue3 := 0;
   B_Pres8.PreviousValue4 := 0;
   B_Pres8.PreviousValue5 := 0;
   B_Pres8.PreviousValue6 := 0;
   B_Pres8.PreviousValue7 := 0;
   B_Pres8.PreviousValue8 := 0;
   B_Pres8.PreviousValue9 := 0;
   B_Pres8.Count := 0;
   B_Pres8.Mean10 := 0;
   B_Pres8.StanDev := 0;
   B_Pres8.State := 0;
   B_Pres8.MeanStart := 0;
END_ROUTINE

ROUTINE Initial_B_Pres9   (* structured text *)
   B_Pres9.CurrentValue := 0;
   B_Pres9.PreviousValue0 := 0;
   B_Pres9.PreviousValue1 := 0;
   B_Pres9.PreviousValue2 := 0;
   B_Pres9.PreviousValue3 := 0;
   B_Pres9.PreviousValue4 := 0;
   B_Pres9.PreviousValue5 := 0;
   B_Pres9.PreviousValue6 := 0;
   B_Pres9.PreviousValue7 := 0;
   B_Pres9.PreviousValue8 := 0;
   B_Pres9.PreviousValue9 := 0;
   B_Pres9.Count := 0;
   B_Pres9.Mean10 := 0;
   B_Pres9.StanDev := 0;
   B_Pres9.State := 0;
   B_Pres9.MeanStart := 0;
END_ROUTINE

ROUTINE Initial_B_Tem0   (* structured text *)
   B_Tem0.CurrentValue := 0;
   B_Tem0.PreviousValue0 := 0;
   B_Tem0.PreviousValue1 := 0;
   B_Tem0.PreviousValue2 := 0;
   B_Tem0.PreviousValue3 := 0;
   B_Tem0.PreviousValue4 := 0;
   B_Tem0.PreviousValue5 := 0;
   B_Tem0.PreviousValue6 := 0;
   B_Tem0.PreviousValue7 := 0;
   B_Tem0.PreviousValue8 := 0;
   B_Tem0.PreviousValue9 := 0;
   B_Tem0.Count := 0;
   B_Tem0.Mean10 := 0;
   B_Tem0.StanDev := 0;
   B_Tem0.State := 0;
   B_Tem0.MeanStart := 0;
END_ROUTINE

ROUTINE Initial_B_Tem1   (* structured text *)
   B_Tem1.CurrentValue := 0;
   B_Tem1.PreviousValue0 := 0;
   B_Tem1.PreviousValue1 := 0;
   B_Tem1.PreviousValue2 := 0;
   B_Tem1.PreviousValue3 := 0;
   B_Tem1.PreviousValue4 := 0;
   B_Tem1.PreviousValue5 := 0;
   B_Tem1.PreviousValue6 := 0;
   B_Tem1.PreviousValue7 := 0;
   B_Tem1.PreviousValue8 := 0;
   B_Tem1.PreviousValue9 := 0;
   B_Tem1.Count := 0;
   B_Tem1.Mean10 := 0;
   B_Tem1.StanDev := 0;
   B_Tem1.State := 0;
   B_Tem1.MeanStart := 0;
END_ROUTINE

ROUTINE Initial_C_Las0   (* structured text *)
   C_Las0.CurrentValue := 0;
   C_Las0.PreviousValue0 := 0;
   C_Las0.PreviousValue1 := 0;
   C_Las0.PreviousValue2 := 0;
   C_Las0.PreviousValue3 := 0;
   C_Las0.PreviousValue4 := 0;
   C_Las0.PreviousValue5 := 0;
   C_Las0.PreviousValue6 := 0;
   C_Las0.PreviousValue7 := 0;
   C_Las0.PreviousValue8 := 0;
   C_Las0.PreviousValue9 := 0;
   C_Las0.Count := 0;
   C_Las0.Mean10 := 0;
   C_Las0.StanDev := 0;
   C_Las0.State := 0;
   C_Las0.MeanStart := 0;
END_ROUTINE

ROUTINE Initial_C_Las1   (* structured text *)
   C_Las1.CurrentValue := 0;
   C_Las1.PreviousValue0 := 0;
   C_Las1.PreviousValue1 := 0;
   C_Las1.PreviousValue2 := 0;
   C_Las1.PreviousValue3 := 0;
   C_Las1.PreviousValue4 := 0;
   C_Las1.PreviousValue5 := 0;
   C_Las1.PreviousValue6 := 0;
   C_Las1.PreviousValue7 := 0;
   C_Las1.PreviousValue8 := 0;
   C_Las1.PreviousValue9 := 0;
   C_Las1.Count := 0;
   C_Las1.Mean10 := 0;
   C_Las1.StanDev := 0;
   C_Las1.State := 0;
   C_Las0.MeanStart := 0;
END_ROUTINE

ROUTINE Initial_P_Pres0   (* structured text *)
   P_Pres0.CurrentValue := 0;
   P_Pres0.PreviousValue0 := 0;
   P_Pres0.PreviousValue1 := 0;
   P_Pres0.PreviousValue2 := 0;
   P_Pres0.PreviousValue3 := 0;
   P_Pres0.PreviousValue4 := 0;
   P_Pres0.PreviousValue5 := 0;
   P_Pres0.PreviousValue6 := 0;
   P_Pres0.PreviousValue7 := 0;
   P_Pres0.PreviousValue8 := 0;
   P_Pres0.PreviousValue9 := 0;
   P_Pres0.Count := 0;
   P_Pres0.Mean10 := 0;
   P_Pres0.StanDev := 0;
   P_Pres0.State := 0;
   P_Pres0.MeanStart := 0;
END_ROUTINE

ROUTINE Initial_P_Pres1   (* structured text *)
   P_Pres1.CurrentValue := 0;
   P_Pres1.PreviousValue0 := 0;
   P_Pres1.PreviousValue1 := 0;
   P_Pres1.PreviousValue2 := 0;
   P_Pres1.PreviousValue3 := 0;
   P_Pres1.PreviousValue4 := 0;
   P_Pres1.PreviousValue5 := 0;
   P_Pres1.PreviousValue6 := 0;
   P_Pres1.PreviousValue7 := 0;
   P_Pres1.PreviousValue8 := 0;
   P_Pres1.PreviousValue9 := 0;
   P_Pres1.Count := 0;
   P_Pres1.Mean10 := 0;
   P_Pres1.StanDev := 0;
   P_Pres1.State := 0;
   P_Pres1.MeanStart := 0;
END_ROUTINE

ROUTINE Initial_P_Pres2   (* structured text *)
   P_Pres2.CurrentValue := 0;
   P_Pres2.PreviousValue0 := 0;
   P_Pres2.PreviousValue1 := 0;
   P_Pres2.PreviousValue2 := 0;
   P_Pres2.PreviousValue3 := 0;
   P_Pres2.PreviousValue4 := 0;
   P_Pres2.PreviousValue5 := 0;
   P_Pres2.PreviousValue6 := 0;
   P_Pres2.PreviousValue7 := 0;
   P_Pres2.PreviousValue8 := 0;
   P_Pres2.PreviousValue9 := 0;
   P_Pres2.Count := 0;
   P_Pres2.Mean10 := 0;
   P_Pres2.StanDev := 0;
   P_Pres2.State := 0;
   P_Pres2.MeanStart := 0;
END_ROUTINE

ROUTINE Initial_P_Pres3   (* structured text *)
   P_Pres3.CurrentValue := 0;
   P_Pres3.PreviousValue0 := 0;
   P_Pres3.PreviousValue1 := 0;
   P_Pres3.PreviousValue2 := 0;
   P_Pres3.PreviousValue3 := 0;
   P_Pres3.PreviousValue4 := 0;
   P_Pres3.PreviousValue5 := 0;
   P_Pres3.PreviousValue6 := 0;
   P_Pres3.PreviousValue7 := 0;
   P_Pres3.PreviousValue8 := 0;
   P_Pres3.PreviousValue9 := 0;
   P_Pres3.Count := 0;
   P_Pres3.Mean10 := 0;
   P_Pres3.StanDev := 0;
   P_Pres3.State := 0;
   P_Pres3.MeanStart := 0;
END_ROUTINE

ROUTINE Initial_P_Pres4   (* structured text *)
   P_Pres4.CurrentValue := 0;
   P_Pres4.PreviousValue0 := 0;
   P_Pres4.PreviousValue1 := 0;
   P_Pres4.PreviousValue2 := 0;
   P_Pres4.PreviousValue3 := 0;
   P_Pres4.PreviousValue4 := 0;
   P_Pres4.PreviousValue5 := 0;
   P_Pres4.PreviousValue6 := 0;
   P_Pres4.PreviousValue7 := 0;
   P_Pres4.PreviousValue8 := 0;
   P_Pres4.PreviousValue9 := 0;
   P_Pres4.Count := 0;
   P_Pres4.Mean10 := 0;
   P_Pres4.StanDev := 0;
   P_Pres4.State := 0;
   P_Pres4.MeanStart := 0;
END_ROUTINE

ROUTINE Initial_P_Tem1   (* structured text *)
   P_Tem1.CurrentValue := 0;
   P_Tem1.PreviousValue0 := 0;
   P_Tem1.PreviousValue1 := 0;
   P_Tem1.PreviousValue2 := 0;
   P_Tem1.PreviousValue3 := 0;
   P_Tem1.PreviousValue4 := 0;
   P_Tem1.PreviousValue5 := 0;
   P_Tem1.PreviousValue6 := 0;
   P_Tem1.PreviousValue7 := 0;
   P_Tem1.PreviousValue8 := 0;
   P_Tem1.PreviousValue9 := 0;
   P_Tem1.Count := 0;
   P_Tem1.Mean10 := 0;
   P_Tem1.StanDev := 0;
   P_Tem1.State := 0;
   P_Tem1.MeanStart := 0;
END_ROUTINE

ROUTINE Initial_P_Tem2   (* structured text *)
   P_Tem2.CurrentValue := 0;
   P_Tem2.PreviousValue0 := 0;
   P_Tem2.PreviousValue1 := 0;
   P_Tem2.PreviousValue2 := 0;
   P_Tem2.PreviousValue3 := 0;
   P_Tem2.PreviousValue4 := 0;
   P_Tem2.PreviousValue5 := 0;
   P_Tem2.PreviousValue6 := 0;
   P_Tem2.PreviousValue7 := 0;
   P_Tem2.PreviousValue8 := 0;
   P_Tem2.PreviousValue9 := 0;
   P_Tem2.Count := 0;
   P_Tem2.Mean10 := 0;
   P_Tem2.StanDev := 0;
   P_Tem2.State := 0;
   P_Tem2.MeanStart := 0;
END_ROUTINE

ROUTINE Initial_P_Tem3   (* structured text *)
   P_Tem3.CurrentValue := 0;
   P_Tem3.PreviousValue0 := 0;
   P_Tem3.PreviousValue1 := 0;
   P_Tem3.PreviousValue2 := 0;
   P_Tem3.PreviousValue3 := 0;
   P_Tem3.PreviousValue4 := 0;
   P_Tem3.PreviousValue5 := 0;
   P_Tem3.PreviousValue6 := 0;
   P_Tem3.PreviousValue7 := 0;
   P_Tem3.PreviousValue8 := 0;
   P_Tem3.PreviousValue9 := 0;
   P_Tem3.Count := 0;
   P_Tem3.Mean10 := 0;
   P_Tem3.StanDev := 0;
   P_Tem3.State := 0;
   P_Tem3.MeanStart := 0;
END_ROUTINE

ROUTINE Initial_P_Tem4   (* structured text *)
   P_Tem4.CurrentValue := 0;
   P_Tem4.PreviousValue0 := 0;
   P_Tem4.PreviousValue1 := 0;
   P_Tem4.PreviousValue2 := 0;
   P_Tem4.PreviousValue3 := 0;
   P_Tem4.PreviousValue4 := 0;
   P_Tem4.PreviousValue5 := 0;
   P_Tem4.PreviousValue6 := 0;
   P_Tem4.PreviousValue7 := 0;
   P_Tem4.PreviousValue8 := 0;
   P_Tem4.PreviousValue9 := 0;
   P_Tem4.Count := 0;
   P_Tem4.Mean10 := 0;
   P_Tem4.StanDev := 0;
   P_Tem4.State := 0;
   P_Tem4.MeanStart := 0;
END_ROUTINE

ROUTINE MainRoutine   (* structured text *)
// The main routine
   if s:fs then
   Initialized := 0;
   end_if;
   
   if Initialized = 5380 then
   JSR(A02_Update); //Update all sensor & state variables
   JSR(A03_Process); //Calculate distance, velocity and acceleration
   JSR(A04_State); //Check the current state of pod
   JSR(A05_Actions); //Based on state, perform respective actions
   else
   JSR(A01_Initialize); //Initializes Program at start up
   end_if;
END_ROUTINE

ROUTINE MiniMax   (* structured text *)
   case STATE of
   	1: B0_Min := 195; B0_Max := 205; B1_Min := 100; B1_Max := 110; B3_Min := 15; B3_Max := 15; P_Min := 250; P_Max := 300;
   	2: B0_Min := 195; B0_Max := 205; B1_Min := 100; B1_Max := 110; B3_Min := 15; B3_Max := 15; P_Min := 250; P_Max := 300;
   	3: B0_Min := 195; B0_Max := 205; B1_Min := 100; B1_Max := 110; B3_Min := 15; B3_Max := 15; P_Min := 250; P_Max := 300;
   	4: B0_Min := 195; B0_Max := 205; B1_Min := 100; B1_Max := 110; B3_Min := 15; B3_Max := 15; P_Min := 0; P_Max := 3000;
   	5: B0_Min := 195; B0_Max := 205; B1_Min := 100; B1_Max := 110; B3_Min := 100; B3_Max := 110; P_Min := 0; P_Max := 300;
   	6: B0_Min := 195; B0_Max := 205; B1_Min := 100; B1_Max := 110; B3_Min := 15; B3_Max := 15; P_Min := 0; P_Max := 300;
   	7: B0_Min := 105; B0_Max := 155; B1_Min := 100; B1_Max := 110; B3_Min := 15; B3_Max := 15; P_Min := 0; P_Max := 300;
   	8: B0_Min := 105; B0_Max := 155; B1_Min := 100; B1_Max := 110; B3_Min := 15; B3_Max := 15; P_Min := 0; P_Max := 300;
   	9: B0_Min := 105; B0_Max := 155; B1_Min := 100; B1_Max := 110; B3_Min := 15; B3_Max := 15; P_Min := 0; P_Max := 300;
   	10: B0_Min := 195; B0_Max := 205; B1_Min := 100; B1_Max := 110; B3_Min := 100; B3_Max := 110; P_Min := 0; P_Max := 300;
   end_case;
END_ROUTINE

ROUTINE NomCheck_B1   (* structured text *)
   if (B_Pres0.CurrentValue > B0_Max) OR (B_Pres0.CurrentValue < B0_Min) then
   		B_Pres0.State := 2;
   else B_Pres0.State := 0;
   end_if;
   if (B_Pres1.CurrentValue > B1_Max) OR (B_Pres1.CurrentValue < B1_Min) then
   		B_Pres1.State := 2;
   else B_Pres1.State := 0;
   end_if;
   if (B_Pres5.CurrentValue > B0_Max) OR (B_Pres5.CurrentValue < B0_Min) then
   		B_Pres5.State := 2;
   else B_Pres5.State := 0;
   end_if;
   if (B_Pres6.CurrentValue > B1_Max) OR (B_Pres6.CurrentValue < B1_Min) then
   		B_Pres6.State := 2;
   else B_Pres6.State := 0;
   end_if;
   if (B_Pres2.CurrentValue > B1_Max) OR (B_Pres2.CurrentValue < B1_Min) then
   		B_Pres2.State := 2;
   else B_Pres2.State := 0;
   end_if;
   if (B_Pres3.CurrentValue > B3_Max) OR (B_Pres3.CurrentValue < B3_Min) then
   		B_Pres3.State := 2;
   else B_Pres3.State := 0;
   end_if;
   if (B_Pres7.CurrentValue > B1_Max) OR (B_Pres7.CurrentValue < B1_Min) then
   		B_Pres7.State := 2;
   else B_Pres7.State := 0;
   end_if;
   if (B_Pres8.CurrentValue > B3_Max) OR (B_Pres8.CurrentValue < B3_Min) then
   		B_Pres8.State := 2;
   else B_Pres8.State := 0;
   end_if;
   if (B_Pres4.CurrentValue > B3_Max) OR (B_Pres4.CurrentValue < B3_Min) then
   		B_Pres4.State := 2;
   else B_Pres4.State := 0;
   end_if;
   if (B_Pres9.CurrentValue > B3_Max) OR (B_Pres9.CurrentValue < B3_Min) then
   		B_Pres9.State := 2;
   else B_Pres9.State := 0;
   end_if;
   if (B_Tem0.CurrentValue > 305) OR (B_Tem0.CurrentValue < 295) then
   		B_Tem0.State := 2;
   else B_Tem0.State := 0;
   end_if;
   if (B_Tem1.CurrentValue > 305) OR (B_Tem1.CurrentValue < 295) then
   		B_Tem1.State := 2;
   else B_Tem1.State := 0;
   end_if;
   B_NomCount := 24 - (B_Pres0.State + B_Pres1.State + B_Pres2.State + B_Pres3.State + B_Pres4.State + B_Pres5.State + B_Pres6.State + B_Pres7.State + B_Pres8.State + B_Pres9.State + B_Tem0.State + B_Tem1.State);
END_ROUTINE

ROUTINE NomCheck_BT   (* structured text *)
   if (BATTERY_TEMP > 333) OR (BATTERY_TEMP < 253) then
   		Bat_Temp_State := 2;
   else Bat_Temp_State := 0;
   end_if;
   if (BATTERY_VOLTAGE > 29) OR (BATTERY_VOLTAGE < 23) then
   		Bat_Volt_State := 2;
   else Bat_Volt_State := 0;
   end_if;
   //if (BATTERY_CURRENT > 10) OR (BATTERY_CURRENT <= 0) then
   //		Bat_Amp_State := 2;
   //else Bat_Amp_State := 0;
   //end_if;
END_ROUTINE

ROUTINE NomCheck_P1   (* structured text *)
   if P_Pres0.CurrentValue > 100 then
   	P_Pres0.State := 2;
   else P_Pres0.State := 0;
   end_if;
   if P_Pres1.CurrentValue > 3000 then
   	P_Pres1.State := 2;
   else P_Pres1.State := 0;
   end_if;
   if P_Pres2.CurrentValue > 3000 then
   	P_Pres2.State := 2;
   else P_Pres2.State := 0;
   end_if;
   if P_Pres3.CurrentValue > 3000 then
   	P_Pres3.State := 2;
   else P_Pres3.State := 0;
   end_if;
   if P_Pres4.CurrentValue > 3000 then
   	P_Pres4.State := 2;
   else P_Pres4.State := 0;
   end_if;
   if (P_Tem1.CurrentValue > 375) OR (P_Tem1.CurrentValue < 170) then
   		P_Tem1.State := 2;
   else P_Tem1.State := 0;
   end_if;
   if (P_Tem2.CurrentValue > 375) OR (P_Tem2.CurrentValue < 170) then
   		P_Tem2.State := 2;
   else P_Tem2.State := 0;
   end_if;
   if (P_Tem3.CurrentValue > 375) OR (P_Tem3.CurrentValue < 170) then
   		P_Tem3.State := 2;
   else P_Tem3.State := 0;
   end_if;
   if (P_Tem4.CurrentValue > 375) OR (P_Tem4.CurrentValue < 170) then
   		P_Tem4.State := 2;
   else P_Tem4.State := 0;
   end_if;
   P_NomCount := 18 - (P_Pres0.State + P_Pres1.State + P_Pres2.State + P_Pres3.State + P_Pres4.State + P_Tem1.State + P_Tem2.State + P_Tem3.State + P_Tem4.State);
END_ROUTINE

ROUTINE Simulate_B_Pres0   (* structured text *)
   /*B_Pres0.CurrentValue := 3500 - CountOfTimerCompletion*60; //3440, 3380,....,0; 60/sec
   TONR(SIMULATOR);
   SIMULATOR.PRE := 1000;
   SIMULATOR.TimerEnable := 1;
   SIMULATOR.Reset := 0;
   
   if SIMULATOR.DN then
   	CTUD(CountOfTimerCompletion);
   	SIMULATOR.Reset := 1;
   end_if;
   */
END_ROUTINE

ROUTINE Update   (* structured text *)
   if READY then
   	P_Pres0.CurrentValue := 250;
   	P_Pres1.CurrentValue := 3500 - count*6;
   	P_Pres2.CurrentValue := 3500 - count*6;
   	P_Pres3.CurrentValue := 3500 - count*6;
   	P_Pres4.CurrentValue := 3500 - count*6;
   	P_Tem0.CurrentValue := 25;
   	P_Tem1.CurrentValue := 25;
   	P_Tem2.CurrentValue := 25;
   	P_Tem3.CurrentValue := 25;
   	P_Tem4.CurrentValue := 25;
   	count := count + 1;
   elsif P_Pres0_FAILURE then
   	P_Pres0.CurrentValue := 255;
   	P_Pres1.CurrentValue := 3500 - count*6;
   	P_Pres2.CurrentValue := 3500 - count*6;
   	P_Pres3.CurrentValue := 3500 - count*6;
   	P_Pres4.CurrentValue := 3500 - count*6;
   	P_Tem0.CurrentValue := 25;
   	P_Tem1.CurrentValue := 25;
   	P_Tem2.CurrentValue := 25;
   	P_Tem3.CurrentValue := 25;
   	P_Tem4.CurrentValue := 25;
   	count := count + 1;
   elsif P_Pres1_FAILURE then
   	P_Pres0.CurrentValue := 250;
   	P_Pres1.CurrentValue := 4000 - count*6;
   	P_Pres2.CurrentValue := 3500 - count*6;
   	P_Pres3.CurrentValue := 3500 - count*6;
   	P_Pres4.CurrentValue := 3500 - count*6;
   	P_Tem0.CurrentValue := 25;
   	P_Tem1.CurrentValue := 25;
   	P_Tem2.CurrentValue := 25;
   	P_Tem3.CurrentValue := 25;
   	P_Tem4.CurrentValue := 25;
   	count := count + 1;
   elsif P_Pres2_FAILURE then
   	P_Pres0.CurrentValue := 250;
   	P_Pres1.CurrentValue := 3500 - count*6;
   	P_Pres2.CurrentValue := 4000 - count*6;
   	P_Pres3.CurrentValue := 3500 - count*6;
   	P_Pres4.CurrentValue := 3500 - count*6;
   	P_Tem0.CurrentValue := 25;
   	P_Tem1.CurrentValue := 25;
   	P_Tem2.CurrentValue := 25;
   	P_Tem3.CurrentValue := 25;
   	P_Tem4.CurrentValue := 25;
   	count := count + 1;
   elsif P_Pres3_FAILURE then
   	P_Pres0.CurrentValue := 250;
   	P_Pres1.CurrentValue := 3500 - count*6;
   	P_Pres2.CurrentValue := 3500 - count*6;
   	P_Pres3.CurrentValue := 4000 - count*6;
   	P_Pres4.CurrentValue := 3500 - count*6;
   	P_Tem0.CurrentValue := 25;
   	P_Tem1.CurrentValue := 25;
   	P_Tem2.CurrentValue := 25;
   	P_Tem3.CurrentValue := 25;
   	P_Tem4.CurrentValue := 25;
   	count := count + 1;
   elsif P_Pres4_FAILURE then
   	P_Pres0.CurrentValue := 250;
   	P_Pres1.CurrentValue := 3500 - count*6;
   	P_Pres2.CurrentValue := 3500 - count*6;
   	P_Pres3.CurrentValue := 3500 - count*6;
   	P_Pres4.CurrentValue := 4000 - count*6;
   	P_Tem0.CurrentValue := 25;
   	P_Tem1.CurrentValue := 25;
   	P_Tem2.CurrentValue := 25;
   	P_Tem3.CurrentValue := 25;
   	P_Tem4.CurrentValue := 25;
   	count := count + 1;
   elsif P_Tem0_FAILURE then
   	P_Pres0.CurrentValue := 250;
   	P_Pres1.CurrentValue := 3500 - count*6;
   	P_Pres2.CurrentValue := 3500 - count*6;
   	P_Pres3.CurrentValue := 3500 - count*6;
   	P_Pres4.CurrentValue := 3500 - count*6;
   	P_Tem0.CurrentValue := 30;
   	P_Tem1.CurrentValue := 25;
   	P_Tem2.CurrentValue := 25;
   	P_Tem3.CurrentValue := 25;
   	P_Tem4.CurrentValue := 25;
   	count := count + 1;
   elsif P_Tem1_FAILURE then
   	P_Pres0.CurrentValue := 250;
   	P_Pres1.CurrentValue := 3500 - count*6;
   	P_Pres2.CurrentValue := 3500 - count*6;
   	P_Pres3.CurrentValue := 3500 - count*6;
   	P_Pres4.CurrentValue := 3500 - count*6;
   	P_Tem0.CurrentValue := 25;
   	P_Tem1.CurrentValue := 30;
   	P_Tem2.CurrentValue := 25;
   	P_Tem3.CurrentValue := 25;
   	P_Tem4.CurrentValue := 25;
   	count := count + 1;
   elsif P_Tem2_FAILURE then
   	P_Pres0.CurrentValue := 250;
   	P_Pres1.CurrentValue := 3500 - count*6;
   	P_Pres2.CurrentValue := 3500 - count*6;
   	P_Pres3.CurrentValue := 3500 - count*6;
   	P_Pres4.CurrentValue := 3500 - count*6;
   	P_Tem0.CurrentValue := 25;
   	P_Tem1.CurrentValue := 25;
   	P_Tem2.CurrentValue := 30;
   	P_Tem3.CurrentValue := 25;
   	P_Tem4.CurrentValue := 25;
   	count := count + 1;
   elsif P_Tem3_FAILURE then
   	P_Pres0.CurrentValue := 250;
   	P_Pres1.CurrentValue := 3500 - count*6;
   	P_Pres2.CurrentValue := 3500 - count*6;
   	P_Pres3.CurrentValue := 3500 - count*6;
   	P_Pres4.CurrentValue := 3500 - count*6;
   	P_Tem0.CurrentValue := 25;
   	P_Tem1.CurrentValue := 25;
   	P_Tem2.CurrentValue := 25;
   	P_Tem3.CurrentValue := 30;
   	P_Tem4.CurrentValue := 25;
   	count := count + 1;
   elsif P_Tem4_FAILURE then
   	P_Pres0.CurrentValue := 250;
   	P_Pres1.CurrentValue := 3500 - count*6;
   	P_Pres2.CurrentValue := 3500 - count*6;
   	P_Pres3.CurrentValue := 3500 - count*6;
   	P_Pres4.CurrentValue := 3500 - count*6;
   	P_Tem0.CurrentValue := 25;
   	P_Tem1.CurrentValue := 25;
   	P_Tem2.CurrentValue := 25;
   	P_Tem3.CurrentValue := 25;
   	P_Tem4.CurrentValue := 30;
   	count := count + 1;
   elsif TOTAL_FAILURE then
   	P_Pres0.CurrentValue := 255;
   	P_Pres1.CurrentValue := 4000 - count*6/1000;
   	P_Pres2.CurrentValue := 4000 - count*6/1000;
   	P_Pres3.CurrentValue := 4000 - count*6/1000;
   	P_Pres4.CurrentValue := 4000 - count*6/1000;
   	P_Tem0.CurrentValue := 30;
   	P_Tem1.CurrentValue := 30;
   	P_Tem2.CurrentValue := 30;
   	P_Tem3.CurrentValue := 30;
   	P_Tem4.CurrentValue := 30;
   	count := count + 1;
   end_if;
   if count > 666000 then
   	count := 0;
   end_if;
END_ROUTINE

ROUTINE Update_B_Pres0   (* structured text *)
// Routine for Brakes Pressure Sensor #0
   case B_Pres0.Count of
   	0: B_Pres0.PreviousValue0 := B_Pres0.CurrentValue;
   	1: B_Pres0.PreviousValue1 := B_Pres0.CurrentValue;
   	2: B_Pres0.PreviousValue2 := B_Pres0.CurrentValue;
   	3: B_Pres0.PreviousValue3 := B_Pres0.CurrentValue;
   	4: B_Pres0.PreviousValue4 := B_Pres0.CurrentValue;
   	5: B_Pres0.PreviousValue5 := B_Pres0.CurrentValue;
   	6: B_Pres0.PreviousValue6 := B_Pres0.CurrentValue;
   	7: B_Pres0.PreviousValue7 := B_Pres0.CurrentValue;
   	8: B_Pres0.PreviousValue8 := B_Pres0.CurrentValue;
   	9: B_Pres0.PreviousValue9 := B_Pres0.CurrentValue;
   end_case;
   B_Pres0.Count := B_Pres0.Count + 1;
   if B_Pres0.Count = 10 then
   	B_Pres0.Count := 0;
   	B_Pres0.MeanStart := 1;
   end_if;
   B_Pres0.CurrentValue := Local:1:I.Ch00.Data;
   if B_Pres0.MeanStart then
   	B_Pres0.Mean10 := (B_Pres0.PreviousValue0 + B_Pres0.PreviousValue1 + B_Pres0.PreviousValue2 + B_Pres0.PreviousValue3 + B_Pres0.PreviousValue4 + B_Pres0.PreviousValue5 + B_Pres0.PreviousValue6 + B_Pres0.PreviousValue7 + B_Pres0.PreviousValue8 + B_Pres0.PreviousValue9)/10;
   	B_Pres0.StanDev := SQRT(((B_Pres0.PreviousValue0 - B_Pres0.Mean10)**2 + (B_Pres0.PreviousValue1 - B_Pres0.Mean10)**2 + (B_Pres0.PreviousValue2 - B_Pres0.Mean10)**2 + (B_Pres0.PreviousValue3 - B_Pres0.Mean10)**2 + (B_Pres0.PreviousValue4 - B_Pres0.Mean10)**2 + (B_Pres0.PreviousValue5 - B_Pres0.Mean10)**2 + (B_Pres0.PreviousValue6 - B_Pres0.Mean10)**2 + (B_Pres0.PreviousValue7 - B_Pres0.Mean10)**2 + (B_Pres0.PreviousValue8 - B_Pres0.Mean10)**2 + (B_Pres0.PreviousValue9 - B_Pres0.Mean10)**2)/10);
   end_if;
END_ROUTINE
